(* Schneider Machine Expert - Basic project OIL_GAS_CRUDE_TRANSFER_COMPLEX_OPENABLE, file version 3.0.0.0 *)
(* ProjectInformations: Name=New project *)

HARDWARE
  Cpu 0: TM221CE24R
  ModuleExtensionObject 0: TM3DI32K
  ModuleExtensionObject 1: TM3AI2H/G
  EthernetConfiguration: NetworkName=M221, IpAllocationMode=FixedAddress, IpAddress=0.0.0.0, SubnetMask=0.0.0.0
  SerialLineConfiguration: Baud=Baud19200, Parity=ParityEven, DataBits=DataBits8, StopBits=StopBits1, PhysicalMedium=PhysicalMediumRs485, TransmissionMode=TransmissionModeModbusRtu, SlaveId=1, Addressing=SlaveAddressing
  MastTask: UsePeriodScanMode=false, PeriodScan=100
  FastTask: Period=255
  CpuBehavior: StartingMode=StartAsPreviousState, AutoSaveRamOnEeprom=true, WatchdogPeriod=250

SYMBOLS  (address, symbol, comment, settings)
  %M0       AUTO_MODE  "1 automatic; 0 manual"
  %M1       START_HMI  "Remote skid start pulse"
  %M2       STOP_HMI  "Remote normal-stop command"
  %M3       AUTO_ENABLE  "Automatic transfer enable"
  %M10      SYSTEM_RUN  "Crude transfer skid run memory"
  %M11      PROCESS_PERMISSIVE  "Combined ESD, fire-gas, stop-loop, and suction permissive"
  %M12      MANUAL_DEMAND  "Manual run demand"
  %M13      AUTO_DEMAND  "Automatic run demand"
  %M14      SLOP_TANK_HH  "Slop tank high-high shutdown/alarm input from HMI or Modbus"
  %M20      SALES_ROUTE_LATCH  "Current batch selected for sales tank"
  %M21      REPROCESS_ROUTE_LATCH  "Current batch selected for reprocess tank"
  %M22      SLOP_ROUTE_LATCH  "Current batch selected for slop tank"
  %M23      ROUTE_SEQUENCE_BUSY  "Analyzer-to-manifold sequence active"
  %M24      DIVERT_ACTIVE  "Diversion valve dwell phase active"
  %M25      SEQUENCE_RESET  "Sequence-complete reset pulse"
  %M30      COMMON_ALARM  "Common process alarm summary"
  %M40      RESET_BATCH_COUNTERS  "Reset all batch counters"
  %M15      ESD_TRIP_LATCH  "Latched emergency shutdown"
  %M26      SALES_VALVE_FAIL  "Sales valve failed to prove open"
  %M27      REPROCESS_VALVE_FAIL  "Reprocess valve failed to prove open"
  %M28      SLOP_VALVE_FAIL  "Slop valve failed to prove open"
  %M29      PUMP_PROOF_FAIL  "Feed pump failed to prove running"
  %M33      EQUIPMENT_ALARM  "Pump and valve proof-failure group"
  %S6       SB_TB1S  "Time base of 1 s generated by an internal clock"
  %S10      SB_IOCOMBUS  "I/O communication is running correctly (1), I/O communication error detected (0)"
  %S13      SB_FIRSTRUN  "Indicates the first controller cycle in RUN mode"
  %TM0      ANALYZER_TRAVEL_TIMER  "Transport delay from crude analyzer to diversion manifold"
  %TM1      DIVERT_DWELL_TIMER  "Selected diversion valve open dwell time"
  %C0       SALES_BATCH_TOTAL  "Completed on-spec crude batches routed to sales"
  %C1       REPROCESS_BATCH_TOTAL  "Completed off-spec batches routed to reprocess"
  %C2       SLOP_BATCH_TOTAL  "Completed rejected batches routed to slop"
  %I0.0     START_PB  "Local skid start pushbutton"
  %I0.1     STOP_LOOP_OK  "Normal stop loop; 1 healthy"
  %I0.2     ESTOP_OK  "Emergency shutdown relay feedback; 1 healthy"
  %I0.3     FIRE_GAS_OK  "Fire and gas shutdown loop; 1 healthy"
  %I0.4     ANALYZER_TRIGGER  "Crude batch at analyzer; rising edge starts route sequence"
  %I0.5     QUALITY_ONSPEC  "Crude quality is within sales specification"
  %I0.6     REPROCESS_SELECT  "Off-spec batch may be routed to reprocess"
  %I0.7     SUCTION_OK  "Feed-pump suction permissive; 1 healthy"
  %I0.8     DISCHARGE_OK  "Discharge pressure permissive; reserved for commissioning"
  %I0.9     PUMP_OL_OK  "Feed-pump overload feedback; reserved for commissioning"
  %I0.10    SDV_OPEN_FB  "Inlet shutdown valve open feedback; reserved for commissioning"
  %I0.11    SALES_VALVE_FB  "Sales valve open feedback; reserved for commissioning"
  %I0.12    REPROCESS_VALVE_FB  "Reprocess valve open feedback; reserved for commissioning"
  %I0.13    SLOP_VALVE_FB  "Slop valve open feedback; reserved for commissioning"
  %Q0.0     CRUDE_FEED_PUMP  "Crude transfer pump contactor or VFD run"
  %Q0.1     VALVE_TO_SALES  "Sales-tank diversion valve"
  %Q0.2     VALVE_TO_REPROCESS  "Reprocess-tank diversion valve"
  %Q0.3     VALVE_TO_SLOP  "Slop-tank diversion valve"
  %Q0.4     BEACON_RUN  "Skid running beacon"
  %Q0.5     BEACON_ALARM  "Common alarm beacon"
  %Q0.6     HORN_COMMON  "Common audible alarm"
  %Q0.7     SDV_INLET  "Inlet shutdown valve solenoid"
  %Q0.8     PANEL_HEALTHY  "PLC and process healthy indication"
  %Q0.9     PLC_HEARTBEAT  "One-second PLC heartbeat"
  %I1.0     SUCTION_PSL_OK  "Suction low-pressure switch healthy"
  %I1.1     DISCH_PSH_OK  "Discharge high-pressure switch healthy"
  %I1.2     LEAK_DETECT_OK  "Hydrocarbon leak detector healthy"
  %I1.3     GAS_DETECT_OK  "Combustible gas detector healthy"
  %I1.4     ESD_RESET_PB  "Physical ESD reset pushbutton"
  %I1.5     PUMP_RUN_FB  "Crude feed-pump running feedback"
  %I1.6     FIRE_PANEL_OK  "Fire and gas panel healthy"
  %I1.7     UPS_OK  "Control-panel UPS healthy"
  %I1.8     FILTER_DP_OK  "Filter differential-pressure switch healthy"
  %I1.9     SALES_TANK_OK  "Sales tank not high-high"
  %I1.10    REPROCESS_TANK_OK  "Reprocess tank not high-high"
  %I1.11    SLOP_TANK_OK  "Slop tank not high-high"
  %I1.12    VFD_READY  "Pump VFD ready"
  %I1.13    MCC_HEALTHY  "Motor control center healthy"
  %I1.14    SPARE_I1_14  "Reserved expansion digital input"
  %I1.15    SPARE_I1_15  "Reserved expansion digital input"
  %I1.16    SPARE_I1_16  "Reserved expansion digital input"
  %I1.17    SPARE_I1_17  "Reserved expansion digital input"
  %I1.18    SPARE_I1_18  "Reserved expansion digital input"
  %I1.19    SPARE_I1_19  "Reserved expansion digital input"
  %I1.20    SPARE_I1_20  "Reserved expansion digital input"
  %I1.21    SPARE_I1_21  "Reserved expansion digital input"
  %I1.22    SPARE_I1_22  "Reserved expansion digital input"
  %I1.23    SPARE_I1_23  "Reserved expansion digital input"
  %I1.24    SPARE_I1_24  "Reserved expansion digital input"
  %I1.25    SPARE_I1_25  "Reserved expansion digital input"
  %I1.26    SPARE_I1_26  "Reserved expansion digital input"
  %I1.27    SPARE_I1_27  "Reserved expansion digital input"
  %I1.28    SPARE_I1_28  "Reserved expansion digital input"
  %I1.29    SPARE_I1_29  "Reserved expansion digital input"
  %I1.30    SPARE_I1_30  "Reserved expansion digital input"
  %I1.31    SPARE_I1_31  "Reserved expansion digital input"
  %IW2.0    LEVEL_RAW  "Sensor level 4-20 mA raw 4000-20000"  [Type=Type_4_20mA, Scope=Scope_Customized, Minimum=4000, Maximum=20000]

POU CRUDE_TRANSFER_COMPLEX_42R_IL
  (* SectionNumber=0 *)

// Rung 0: N00_BATCH_COUNTER_PRESETS
// First scan: initialize sales, reprocess, and slop batch counter presets.
  LD %S13                 (* SB_FIRSTRUN *)
  [ %C0.P := 9999 ]       (* SALES_BATCH_TOTAL *)
  [ %C1.P := 9999 ]       (* REPROCESS_BATCH_TOTAL *)
  [ %C2.P := 9999 ]       (* SLOP_BATCH_TOTAL *)
  // as ST:
  //   IF SB_FIRSTRUN THEN SALES_BATCH_TOTAL.P := 9999; END_IF;
  //   IF SB_FIRSTRUN THEN REPROCESS_BATCH_TOTAL.P := 9999; END_IF;
  //   IF SB_FIRSTRUN THEN SLOP_BATCH_TOTAL.P := 9999; END_IF;

// Rung 1: N01_COMPLEX_PERMISSIVE
// Stop loop, E-Stop, fire-gas, suction, discharge, expansion safety inputs, HMI stop, and ESD latch.
  LD %I0.1                (* STOP_LOOP_OK *)
  AND %I0.2               (* ESTOP_OK *)
  AND %I0.3               (* FIRE_GAS_OK *)
  AND %I0.7               (* SUCTION_OK *)
  AND %I0.8               (* DISCHARGE_OK *)
  AND %I0.9               (* PUMP_OL_OK *)
  AND %I1.0               (* SUCTION_PSL_OK *)
  AND %I1.1               (* DISCH_PSH_OK *)
  AND %I1.2               (* LEAK_DETECT_OK *)
  AND %I1.3               (* GAS_DETECT_OK *)
  ANDN %M2                (* STOP_HMI *)
  ANDN %M15               (* ESD_TRIP_LATCH *)
  ST %M11                 (* PROCESS_PERMISSIVE *)
  // as ST:
  //   PROCESS_PERMISSIVE := STOP_LOOP_OK AND ESTOP_OK AND FIRE_GAS_OK AND SUCTION_OK AND DISCHARGE_OK AND PUMP_OL_OK AND SUCTION_PSL_OK AND DISCH_PSH_OK AND LEAK_DETECT_OK AND GAS_DETECT_OK AND NOT STOP_HMI AND NOT ESD_TRIP_LATCH;

// Rung 2: N02_MANUAL_START_DEMAND
// Local or HMI start demand in manual mode; retain demand while the skid is running.
  LD %I0.0                (* START_PB *)
  OR %M1                  (* START_HMI *)
  OR %M10                 (* SYSTEM_RUN *)
  ANDN %M0                (* AUTO_MODE *)
  ST %M12                 (* MANUAL_DEMAND *)
  // as ST:
  //   MANUAL_DEMAND := (START_PB OR START_HMI OR SYSTEM_RUN) AND NOT AUTO_MODE;

// Rung 3: N03_AUTO_START_DEMAND
// Automatic start demand when AUTO mode and AUTO enable are active.
  LD %M0                  (* AUTO_MODE *)
  AND %M3                 (* AUTO_ENABLE *)
  ST %M13                 (* AUTO_DEMAND *)
  // as ST:
  //   AUTO_DEMAND := AUTO_MODE AND AUTO_ENABLE;

// Rung 4: N04_SYSTEM_RUN_LATCH
// Run memory is allowed only while all process and safety permissives remain healthy.
  LD %M12                 (* MANUAL_DEMAND *)
  OR %M13                 (* AUTO_DEMAND *)
  AND %M11                (* PROCESS_PERMISSIVE *)
  ST %M10                 (* SYSTEM_RUN *)
  // as ST:
  //   SYSTEM_RUN := (MANUAL_DEMAND OR AUTO_DEMAND) AND PROCESS_PERMISSIVE;

// Rung 5: N05_LATCH_SALES_ROUTE
// At analyzer trigger, latch a sales-tank route when the crude quality input is on-spec.
  LDR %I0.4               (* ANALYZER_TRIGGER *)
  AND %M10                (* SYSTEM_RUN *)
  ANDN %M23               (* ROUTE_SEQUENCE_BUSY *)
  AND %I0.5               (* QUALITY_ONSPEC *)
  S %M20                  (* SALES_ROUTE_LATCH *)
  // as ST:
  //   IF RISING(ANALYZER_TRIGGER) AND SYSTEM_RUN AND NOT ROUTE_SEQUENCE_BUSY AND QUALITY_ONSPEC THEN SALES_ROUTE_LATCH := TRUE; END_IF;

// Rung 6: N06_LATCH_REPROCESS_ROUTE
// Latch reprocess route when quality is off-spec but the reprocess selector is active.
  LDR %I0.4               (* ANALYZER_TRIGGER *)
  AND %M10                (* SYSTEM_RUN *)
  ANDN %M23               (* ROUTE_SEQUENCE_BUSY *)
  ANDN %I0.5              (* QUALITY_ONSPEC *)
  AND %I0.6               (* REPROCESS_SELECT *)
  S %M21                  (* REPROCESS_ROUTE_LATCH *)
  // as ST:
  //   IF RISING(ANALYZER_TRIGGER) AND SYSTEM_RUN AND NOT ROUTE_SEQUENCE_BUSY AND NOT QUALITY_ONSPEC AND REPROCESS_SELECT THEN REPROCESS_ROUTE_LATCH := TRUE; END_IF;

// Rung 7: N07_LATCH_SLOP_ROUTE
// Latch slop route when neither sales nor reprocess quality condition is selected.
  LDR %I0.4               (* ANALYZER_TRIGGER *)
  AND %M10                (* SYSTEM_RUN *)
  ANDN %M23               (* ROUTE_SEQUENCE_BUSY *)
  ANDN %I0.5              (* QUALITY_ONSPEC *)
  ANDN %I0.6              (* REPROCESS_SELECT *)
  S %M22                  (* SLOP_ROUTE_LATCH *)
  // as ST:
  //   IF RISING(ANALYZER_TRIGGER) AND SYSTEM_RUN AND NOT ROUTE_SEQUENCE_BUSY AND NOT QUALITY_ONSPEC AND NOT REPROCESS_SELECT THEN SLOP_ROUTE_LATCH := TRUE; END_IF;

// Rung 8: N08_ROUTE_SEQUENCE_BUSY
// Prevent a second analyzer trigger while the current diversion sequence is active.
  LDR %I0.4               (* ANALYZER_TRIGGER *)
  AND %M10                (* SYSTEM_RUN *)
  ANDN %M23               (* ROUTE_SEQUENCE_BUSY *)
  S %M23                  (* ROUTE_SEQUENCE_BUSY *)
  // as ST:
  //   IF RISING(ANALYZER_TRIGGER) AND SYSTEM_RUN AND NOT ROUTE_SEQUENCE_BUSY THEN ROUTE_SEQUENCE_BUSY := TRUE; END_IF;

// Rung 9: N09_ANALYZER_TO_MANIFOLD_TIMER
// Compensate transport time between the crude analyzer and the diversion manifold.
  BLK %TM0                (* ANALYZER_TRAVEL_TIMER *)
  LD %M23                 (* ROUTE_SEQUENCE_BUSY *)
  ANDN %M24               (* DIVERT_ACTIVE *)
  IN
  END_BLK
  // as ST:
  //   ANALYZER_TRAVEL_TIMER(IN := ROUTE_SEQUENCE_BUSY AND NOT DIVERT_ACTIVE);

// Rung 10: N10_ENABLE_DIVERT_PHASE
// Start the physical diversion phase after the transport delay expires.
  LD %TM0.Q               (* ANALYZER_TRAVEL_TIMER *)
  S %M24                  (* DIVERT_ACTIVE *)
  // as ST:
  //   IF ANALYZER_TRAVEL_TIMER.Q THEN DIVERT_ACTIVE := TRUE; END_IF;

// Rung 11: N11_DIVERT_VALVE_DWELL_TIMER
// Hold the selected diversion valve open for the configured dwell time.
  BLK %TM1                (* DIVERT_DWELL_TIMER *)
  LD %M24                 (* DIVERT_ACTIVE *)
  IN
  END_BLK
  // as ST:
  //   DIVERT_DWELL_TIMER(IN := DIVERT_ACTIVE);

// Rung 12: N12_COMPLEX_FEED_PUMP
// Crude feed pump requires run memory, complete permissive, discharge/suction health, and no diversion phase.
  LD %M10                 (* SYSTEM_RUN *)
  AND %M11                (* PROCESS_PERMISSIVE *)
  ANDN %M24               (* DIVERT_ACTIVE *)
  ANDN %M14               (* SLOP_TANK_HH *)
  AND %I0.8               (* DISCHARGE_OK *)
  AND %I0.9               (* PUMP_OL_OK *)
  ST %Q0.0                (* CRUDE_FEED_PUMP *)
  // as ST:
  //   CRUDE_FEED_PUMP := SYSTEM_RUN AND PROCESS_PERMISSIVE AND NOT DIVERT_ACTIVE AND NOT SLOP_TANK_HH AND DISCHARGE_OK AND PUMP_OL_OK;

// Rung 13: N13_SALES_VALVE
// Open the sales-tank valve for an on-spec batch during the diversion phase.
  LD %M24                 (* DIVERT_ACTIVE *)
  AND %M20                (* SALES_ROUTE_LATCH *)
  AND %M11                (* PROCESS_PERMISSIVE *)
  ST %Q0.1                (* VALVE_TO_SALES *)
  // as ST:
  //   VALVE_TO_SALES := DIVERT_ACTIVE AND SALES_ROUTE_LATCH AND PROCESS_PERMISSIVE;

// Rung 14: N14_REPROCESS_VALVE
// Open the reprocess valve for a recoverable off-spec batch.
  LD %M24                 (* DIVERT_ACTIVE *)
  AND %M21                (* REPROCESS_ROUTE_LATCH *)
  AND %M11                (* PROCESS_PERMISSIVE *)
  ST %Q0.2                (* VALVE_TO_REPROCESS *)
  // as ST:
  //   VALVE_TO_REPROCESS := DIVERT_ACTIVE AND REPROCESS_ROUTE_LATCH AND PROCESS_PERMISSIVE;

// Rung 15: N15_SLOP_VALVE
// Open the slop valve for a rejected off-spec batch.
  LD %M24                 (* DIVERT_ACTIVE *)
  AND %M22                (* SLOP_ROUTE_LATCH *)
  AND %M11                (* PROCESS_PERMISSIVE *)
  ST %Q0.3                (* VALVE_TO_SLOP *)
  // as ST:
  //   VALVE_TO_SLOP := DIVERT_ACTIVE AND SLOP_ROUTE_LATCH AND PROCESS_PERMISSIVE;

// Rung 16: N16_COUNT_SALES_BATCH
// Count completed on-spec batches; reset from the counter-reset command.
  BLK %C0                 (* SALES_BATCH_TOTAL *)
  LD %M40                 (* RESET_BATCH_COUNTERS *)
  R
  LD %TM1.Q               (* DIVERT_DWELL_TIMER *)
  AND %M20                (* SALES_ROUTE_LATCH *)
  CU
  END_BLK
  // as ST:
  //   SALES_BATCH_TOTAL(R := RESET_BATCH_COUNTERS, CU := DIVERT_DWELL_TIMER.Q AND SALES_ROUTE_LATCH);

// Rung 17: N17_COUNT_REPROCESS_BATCH
// Count completed reprocess batches; reset from the counter-reset command.
  BLK %C1                 (* REPROCESS_BATCH_TOTAL *)
  LD %M40                 (* RESET_BATCH_COUNTERS *)
  R
  LD %TM1.Q               (* DIVERT_DWELL_TIMER *)
  AND %M21                (* REPROCESS_ROUTE_LATCH *)
  CU
  END_BLK
  // as ST:
  //   REPROCESS_BATCH_TOTAL(R := RESET_BATCH_COUNTERS, CU := DIVERT_DWELL_TIMER.Q AND REPROCESS_ROUTE_LATCH);

// Rung 18: N18_COUNT_SLOP_BATCH
// Count completed slop batches; reset from the counter-reset command.
  BLK %C2                 (* SLOP_BATCH_TOTAL *)
  LD %M40                 (* RESET_BATCH_COUNTERS *)
  R
  LD %TM1.Q               (* DIVERT_DWELL_TIMER *)
  AND %M22                (* SLOP_ROUTE_LATCH *)
  CU
  END_BLK
  // as ST:
  //   SLOP_BATCH_TOTAL(R := RESET_BATCH_COUNTERS, CU := DIVERT_DWELL_TIMER.Q AND SLOP_ROUTE_LATCH);

// Rung 19: N19_SEQUENCE_RESET_PULSE
// Create a sequence reset pulse after valve dwell is complete.
  LD %TM1.Q               (* DIVERT_DWELL_TIMER *)
  ST %M25                 (* SEQUENCE_RESET *)
  // as ST:
  //   SEQUENCE_RESET := DIVERT_DWELL_TIMER.Q;

// Rung 20: N20_RESET_DIVERT_ACTIVE
// Clear the diversion-active state at sequence completion.
  LD %M25                 (* SEQUENCE_RESET *)
  R %M24                  (* DIVERT_ACTIVE *)
  // as ST:
  //   IF SEQUENCE_RESET THEN DIVERT_ACTIVE := FALSE; END_IF;

// Rung 21: N21_RESET_ROUTE_BUSY
// Clear the sequence-busy state at sequence completion.
  LD %M25                 (* SEQUENCE_RESET *)
  R %M23                  (* ROUTE_SEQUENCE_BUSY *)
  // as ST:
  //   IF SEQUENCE_RESET THEN ROUTE_SEQUENCE_BUSY := FALSE; END_IF;

// Rung 22: N22_RESET_SALES_LATCH
// Clear the sales-route latch at sequence completion.
  LD %M25                 (* SEQUENCE_RESET *)
  R %M20                  (* SALES_ROUTE_LATCH *)
  // as ST:
  //   IF SEQUENCE_RESET THEN SALES_ROUTE_LATCH := FALSE; END_IF;

// Rung 23: N23_RESET_REPROCESS_LATCH
// Clear the reprocess-route latch at sequence completion.
  LD %M25                 (* SEQUENCE_RESET *)
  R %M21                  (* REPROCESS_ROUTE_LATCH *)
  // as ST:
  //   IF SEQUENCE_RESET THEN REPROCESS_ROUTE_LATCH := FALSE; END_IF;

// Rung 24: N24_RESET_SLOP_LATCH
// Clear the slop-route latch at sequence completion.
  LD %M25                 (* SEQUENCE_RESET *)
  R %M22                  (* SLOP_ROUTE_LATCH *)
  // as ST:
  //   IF SEQUENCE_RESET THEN SLOP_ROUTE_LATCH := FALSE; END_IF;

// Rung 25: N25_COMMON_ALARM
// Generate common alarm if a process permissive is lost or the slop tank is high-high.
  LDN %M11                (* PROCESS_PERMISSIVE *)
  OR %M14                 (* SLOP_TANK_HH *)
  ST %M30                 (* COMMON_ALARM *)
  // as ST:
  //   COMMON_ALARM := NOT PROCESS_PERMISSIVE OR SLOP_TANK_HH;

// Rung 26: N26_RUN_BEACON
// Energize the run beacon while the skid runs without a common alarm.
  LD %M10                 (* SYSTEM_RUN *)
  ANDN %M30               (* COMMON_ALARM *)
  ST %Q0.4                (* BEACON_RUN *)
  // as ST:
  //   BEACON_RUN := SYSTEM_RUN AND NOT COMMON_ALARM;

// Rung 27: N27_ALARM_BEACON
// Energize the alarm beacon whenever the common alarm is active.
  LD %M30                 (* COMMON_ALARM *)
  ST %Q0.5                (* BEACON_ALARM *)
  // as ST:
  //   BEACON_ALARM := COMMON_ALARM;

// Rung 28: N28_ESTOP_TRIP
// Latch ESD when emergency-stop relay feedback is lost.
  LDN %I0.2               (* ESTOP_OK *)
  S %M15                  (* ESD_TRIP_LATCH *)
  // as ST:
  //   IF NOT ESTOP_OK THEN ESD_TRIP_LATCH := TRUE; END_IF;

// Rung 29: N29_FIRE_GAS_TRIP
// Latch ESD when the primary fire and gas loop is lost.
  LDN %I0.3               (* FIRE_GAS_OK *)
  S %M15                  (* ESD_TRIP_LATCH *)
  // as ST:
  //   IF NOT FIRE_GAS_OK THEN ESD_TRIP_LATCH := TRUE; END_IF;

// Rung 30: N30_LEAK_TRIP
// Latch ESD when the expansion leak-detection loop is lost.
  LDN %I1.2               (* LEAK_DETECT_OK *)
  S %M15                  (* ESD_TRIP_LATCH *)
  // as ST:
  //   IF NOT LEAK_DETECT_OK THEN ESD_TRIP_LATCH := TRUE; END_IF;

// Rung 31: N31_ESD_RESET
// Reset ESD only by physical reset while safety loops are healthy.
  LD %I1.4                (* ESD_RESET_PB *)
  AND %I0.2               (* ESTOP_OK *)
  AND %I0.3               (* FIRE_GAS_OK *)
  AND %I1.2               (* LEAK_DETECT_OK *)
  R %M15                  (* ESD_TRIP_LATCH *)
  // as ST:
  //   IF ESD_RESET_PB AND ESTOP_OK AND FIRE_GAS_OK AND LEAK_DETECT_OK THEN ESD_TRIP_LATCH := FALSE; END_IF;

// Rung 32: N32_PUMP_PROOF_FAIL
// Detect feed-pump command without running feedback.
  LD %Q0.0                (* CRUDE_FEED_PUMP *)
  ANDN %I1.5              (* PUMP_RUN_FB *)
  ST %M29                 (* PUMP_PROOF_FAIL *)
  // as ST:
  //   PUMP_PROOF_FAIL := CRUDE_FEED_PUMP AND NOT PUMP_RUN_FB;

// Rung 33: N33_SALES_VALVE_FAIL
// Detect sales valve command without open feedback.
  LD %Q0.1                (* VALVE_TO_SALES *)
  ANDN %I0.11             (* SALES_VALVE_FB *)
  ST %M26                 (* SALES_VALVE_FAIL *)
  // as ST:
  //   SALES_VALVE_FAIL := VALVE_TO_SALES AND NOT SALES_VALVE_FB;

// Rung 34: N34_REPROCESS_VALVE_FAIL
// Detect reprocess valve command without open feedback.
  LD %Q0.2                (* VALVE_TO_REPROCESS *)
  ANDN %I0.12             (* REPROCESS_VALVE_FB *)
  ST %M27                 (* REPROCESS_VALVE_FAIL *)
  // as ST:
  //   REPROCESS_VALVE_FAIL := VALVE_TO_REPROCESS AND NOT REPROCESS_VALVE_FB;

// Rung 35: N35_SLOP_VALVE_FAIL
// Detect slop valve command without open feedback.
  LD %Q0.3                (* VALVE_TO_SLOP *)
  ANDN %I0.13             (* SLOP_VALVE_FB *)
  ST %M28                 (* SLOP_VALVE_FAIL *)
  // as ST:
  //   SLOP_VALVE_FAIL := VALVE_TO_SLOP AND NOT SLOP_VALVE_FB;

// Rung 36: N36_EQUIPMENT_ALARM
// Group pump and diversion valve proof failures.
  LD %M29                 (* PUMP_PROOF_FAIL *)
  OR %M26                 (* SALES_VALVE_FAIL *)
  OR %M27                 (* REPROCESS_VALVE_FAIL *)
  OR %M28                 (* SLOP_VALVE_FAIL *)
  ST %M33                 (* EQUIPMENT_ALARM *)
  // as ST:
  //   EQUIPMENT_ALARM := PUMP_PROOF_FAIL OR SALES_VALVE_FAIL OR REPROCESS_VALVE_FAIL OR SLOP_VALVE_FAIL;

// Rung 37: N37_COMPLEX_ALARM
// Combine base alarm, ESD latch, equipment alarm, and I/O bus fault.
  LDN %M11                (* PROCESS_PERMISSIVE *)
  OR %M15                 (* ESD_TRIP_LATCH *)
  OR %M33                 (* EQUIPMENT_ALARM *)
  ORN %S10                (* SB_IOCOMBUS *)
  ST %M30                 (* COMMON_ALARM *)
  // as ST:
  //   COMMON_ALARM := NOT PROCESS_PERMISSIVE OR ESD_TRIP_LATCH OR EQUIPMENT_ALARM OR NOT SB_IOCOMBUS;

// Rung 38: N38_COMMON_HORN
// Drive common audible alarm.
  LD %M30                 (* COMMON_ALARM *)
  ST %Q0.6                (* HORN_COMMON *)
  // as ST:
  //   HORN_COMMON := COMMON_ALARM;

// Rung 39: N39_INLET_SDV
// Open inlet shutdown valve only while core safety loops are healthy.
  LD %I0.1                (* STOP_LOOP_OK *)
  AND %I0.2               (* ESTOP_OK *)
  AND %I0.3               (* FIRE_GAS_OK *)
  AND %I1.2               (* LEAK_DETECT_OK *)
  ANDN %M15               (* ESD_TRIP_LATCH *)
  ST %Q0.7                (* SDV_INLET *)
  // as ST:
  //   SDV_INLET := STOP_LOOP_OK AND ESTOP_OK AND FIRE_GAS_OK AND LEAK_DETECT_OK AND NOT ESD_TRIP_LATCH;

// Rung 40: N40_PANEL_HEALTHY
// Indicate healthy PLC and process state.
  LD %S10                 (* SB_IOCOMBUS *)
  AND %M11                (* PROCESS_PERMISSIVE *)
  ANDN %M30               (* COMMON_ALARM *)
  ST %Q0.8                (* PANEL_HEALTHY *)
  // as ST:
  //   PANEL_HEALTHY := SB_IOCOMBUS AND PROCESS_PERMISSIVE AND NOT COMMON_ALARM;

// Rung 41: N41_PLC_HEARTBEAT
// Provide a one-second heartbeat to external monitoring.
  LD %S6                  (* SB_TB1S *)
  ST %Q0.9                (* PLC_HEARTBEAT *)
  // as ST:
  //   PLC_HEARTBEAT := SB_TB1S;
